// TIA Portal V18 export
TYPE "typeGuideAxisInt"
// stored: IsFailsafeCompliant false
   STRUCT
      Mot1_RightLeft : Int;
      Mot2_FwdRev : Int;
   END_STRUCT;
END_TYPE
